INTERFACE ITF_ObslugaAlarmow_ElementWykonawczy

METHOD ZwrocTabliceAktywnychZdarzen : BOOL
VAR_INPUT
END_VAR
END_METHOD

METHOD ZwrocTabliceDefinicjiZdarzen : BOOL
VAR_INPUT
END_VAR
END_METHOD

END_INTERFACE

(* stored: Version 1.1.0.1, ProductVersion 3.1.4024.11
   Itf ITF_ObslugaAlarmow_ElementWykonawczy: Id {ffe17445-c3c0-4eb2-a673-e4455b28cc12}
   Method ZwrocTabliceAktywnychZdarzen: Id {da3b91b4-33cd-4264-a465-2ae530f68d4b}
   Method ZwrocTabliceDefinicjiZdarzen: Id {5c970a7c-f503-45f8-8a34-d6eff132f24e} *)
